(* LS Electric XG5000 project: 미니공정설계 *)
(* PLC LSPLC *)

PROGRAM NewProgram (* task: 스캔 프로그램 *)
VAR
    DELAYTIME : BOOL;
    INST : TMR;
    OPENCV1 AT %MX2 : BOOL;
    RUN AT %MX10 : BOOL;
    START AT %MX0 : BOOL;
    STOP AT %MX1 : BOOL;
END_VAR

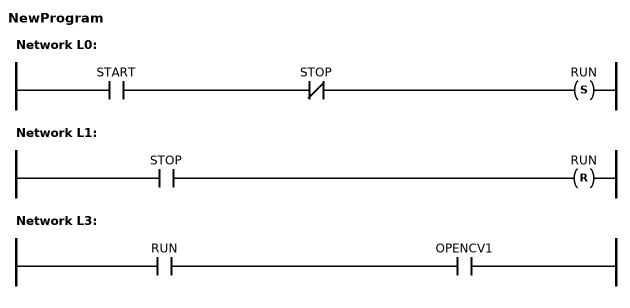
(* Rung L0 *)
IF START AND NOT STOP THEN RUN := TRUE; END_IF;
(* Rung L1 *)
IF STOP THEN RUN := FALSE; END_IF;
(* Rung L3 *)
(* not connected or not rendered: RUN, OPENCV1 *)
END_PROGRAM